// TIA Portal project "Organizador de Cajas" (V18)

(* hardware
DEVICE "S7-1200 station_1"  S7-1200 Station
   slot 0: "Rack_0"  S7-1200 Rack  Rack  V1.0
   slot 1: "PLC_1"  CPU 1212C DC/DC/Rly  6ES7 212-1HE40-0XB0  V4.6
*)

// ===== PLC "PLC_1"  CPU 1212C DC/DC/Rly =====

VAR_GLOBAL   // PLC tag table "Default tag table"
   "pulsadorStart" AT %I0.0 : Bool;
   "pulsadorStop" AT %I0.1 : Bool;
   "setaEmergencia" AT %I0.2 : Bool;
   "infrarrojoEntradaCinta" AT %I0.3 : Bool;
   "infrarrojoPrimerDesviador" AT %I0.4 : Bool;
   "infrarrojoSegundoDesviador" AT %I0.5 : Bool;
   "infrarrojoTercerDesviador" AT %I0.6 : Bool;
   "marcaEnServicio" AT %M90.0 : Bool;
   "marcaPaqueteCinta" AT %M90.1 : Bool;
   "marcaTurnoDesviadorUno" AT %M90.2 : Bool;
   "marcaTurnoDesviadorDos" AT %M90.3 : Bool;
   "marcaTurnoDesviadorTres" AT %M90.4 : Bool;
   "ledStart" AT %Q0.0 : Bool;
   "ledStop" AT %Q0.1 : Bool;
   "motorCintaPrincipal" AT %Q0.2 : Bool;
   "desviadorUno" AT %Q0.3 : Bool;
   "cintaDesviadorUno" AT %Q0.4 : Bool;
   "desviadorDos" AT %Q0.5 : Bool;
   "cintaDesviadorDos" AT %Q0.6 : Bool;
   "desviadorTres" AT %Q0.7 : Bool;
   "cintaDesviadorTres" AT %Q1.0 : Bool;
END_VAR

// folder: System blocks/Program resources

DATA_BLOCK "retardoArranqueCinta"   // DB1
{ S7_Optimized_Access := 'TRUE' }
AUTHOR : Simatic
FAMILY : IEC
NAME : IEC_TMR
VERSION : 1.0
// stored: InstanceOfName IEC_TIMER
"IEC_TIMER"
BEGIN
END_DATA_BLOCK

DATA_BLOCK "cajaSeleccionada"   // DB2
{ S7_Optimized_Access := 'TRUE' }
AUTHOR : Simatic
FAMILY : IEC
NAME : IEC_TMR
VERSION : 1.0
// stored: InstanceOfName IEC_TIMER
"IEC_TIMER"
BEGIN
END_DATA_BLOCK

DATA_BLOCK "CTUDesviadorUno"   // DB3
{ S7_Optimized_Access := 'TRUE' }
AUTHOR : Simatic
FAMILY : IEC
NAME : CNTR
VERSION : 1.0
// stored: InstanceOfName IEC_COUNTER
"IEC_COUNTER"
BEGIN
END_DATA_BLOCK

DATA_BLOCK "CTUDesviadorDos"   // DB4
{ S7_Optimized_Access := 'TRUE' }
AUTHOR : Simatic
FAMILY : IEC
NAME : CNTR
VERSION : 1.0
// stored: InstanceOfName IEC_COUNTER
"IEC_COUNTER"
BEGIN
END_DATA_BLOCK

DATA_BLOCK "CTUDesviadorTres"   // DB5
{ S7_Optimized_Access := 'TRUE' }
AUTHOR : Simatic
FAMILY : IEC
NAME : CNTR
VERSION : 1.0
// stored: InstanceOfName IEC_COUNTER
"IEC_COUNTER"
BEGIN
END_DATA_BLOCK

// folder: (top level)

ORGANIZATION_BLOCK "Main"   // OB1, LAD, ProgramCycle
TITLE = "Main Program Sweep (Cycle)"
{ S7_Optimized_Access := 'TRUE' }
VERSION : 0.1
   VAR_INPUT
      Initial_Call : Bool;   // Initial call of this OB
      Remanence : Bool;   // =True, if remanent data are available
   END_VAR
BEGIN

REGION Network 1: Instalación activa
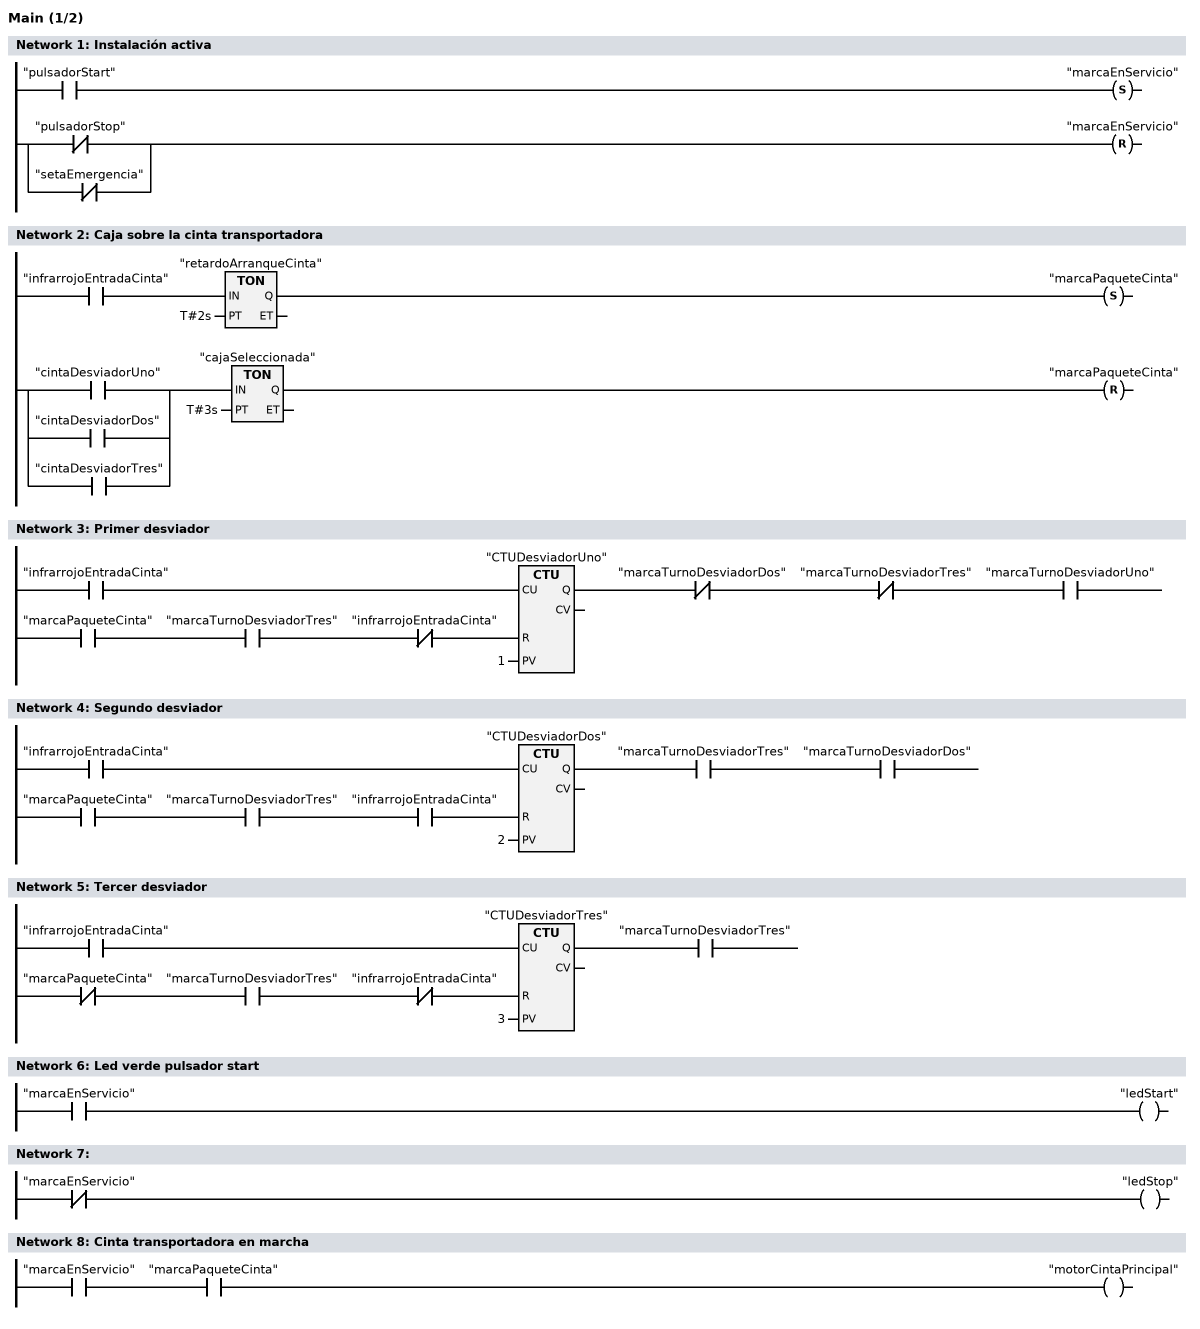
   RUNG wire#powerrail
      Contact( "pulsadorStart" )
      S_Coil( "marcaEnServicio" )
   END_RUNG
   RUNG wire#powerrail
      I_Contact( "pulsadorStop" )
      wire#w1
      R_Coil( "marcaEnServicio" )
   END_RUNG
   RUNG wire#powerrail
      I_Contact( "setaEmergencia" )
   END_RUNG wire#w1
   // the same network as SCL:
   IF "pulsadorStart" THEN "marcaEnServicio" := TRUE; END_IF;
   IF NOT "pulsadorStop" OR NOT "setaEmergencia" THEN "marcaEnServicio" := FALSE; END_IF;
END_REGION

REGION Network 2: Caja sobre la cinta transportadora
   "retardoArranqueCinta".TON(IN := "infrarrojoEntradaCinta", PT := T#2s);
   IF "retardoArranqueCinta".Q THEN "marcaPaqueteCinta" := TRUE; END_IF;
   "cajaSeleccionada".TON(IN := "cintaDesviadorUno" OR "cintaDesviadorDos" OR "cintaDesviadorTres", PT := T#3s);
   IF "cajaSeleccionada".Q THEN "marcaPaqueteCinta" := FALSE; END_IF;
END_REGION

REGION Network 3: Primer desviador
   "CTUDesviadorUno".CTU(CU := "infrarrojoEntradaCinta",
                         R := "marcaPaqueteCinta" AND "marcaTurnoDesviadorTres" AND NOT "infrarrojoEntradaCinta",
                         PV := 1);
END_REGION

REGION Network 4: Segundo desviador
   "CTUDesviadorDos".CTU(CU := "infrarrojoEntradaCinta",
                         R := "marcaPaqueteCinta" AND "marcaTurnoDesviadorTres" AND "infrarrojoEntradaCinta",
                         PV := 2);
END_REGION

REGION Network 5: Tercer desviador
   "CTUDesviadorTres".CTU(CU := "infrarrojoEntradaCinta",
                          R := NOT "marcaPaqueteCinta" AND "marcaTurnoDesviadorTres" AND NOT "infrarrojoEntradaCinta",
                          PV := 3);
END_REGION

REGION Network 6: Led verde pulsador start
   RUNG wire#powerrail
      Contact( "marcaEnServicio" )
      Coil( "ledStart" )
   END_RUNG
   // the same network as SCL:
   "ledStart" := "marcaEnServicio";
END_REGION

REGION Network 7
   RUNG wire#powerrail
      I_Contact( "marcaEnServicio" )
      Coil( "ledStop" )
   END_RUNG
   // the same network as SCL:
   "ledStop" := NOT "marcaEnServicio";
END_REGION

REGION Network 8: Cinta transportadora en marcha
   RUNG wire#powerrail
      Contact( "marcaEnServicio" )
      Contact( "marcaPaqueteCinta" )
      Coil( "motorCintaPrincipal" )
   END_RUNG
   // the same network as SCL:
   "motorCintaPrincipal" := "marcaEnServicio" AND "marcaPaqueteCinta";
END_REGION

REGION Network 9: Desviador uno abierto (accionado) + cinta en marcha
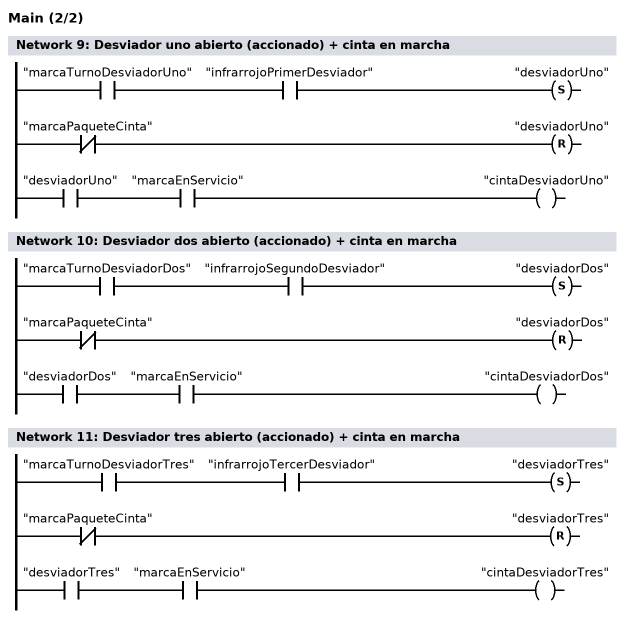
   RUNG wire#powerrail
      Contact( "marcaTurnoDesviadorUno" )
      Contact( "infrarrojoPrimerDesviador" )
      S_Coil( "desviadorUno" )
   END_RUNG
   RUNG wire#powerrail
      I_Contact( "marcaPaqueteCinta" )
      R_Coil( "desviadorUno" )
   END_RUNG
   RUNG wire#powerrail
      Contact( "desviadorUno" )
      Contact( "marcaEnServicio" )
      Coil( "cintaDesviadorUno" )
   END_RUNG
   // the same network as SCL:
   IF "marcaTurnoDesviadorUno" AND "infrarrojoPrimerDesviador" THEN "desviadorUno" := TRUE; END_IF;
   IF NOT "marcaPaqueteCinta" THEN "desviadorUno" := FALSE; END_IF;
   "cintaDesviadorUno" := "desviadorUno" AND "marcaEnServicio";
END_REGION

REGION Network 10: Desviador dos abierto (accionado) + cinta en marcha
   RUNG wire#powerrail
      Contact( "marcaTurnoDesviadorDos" )
      Contact( "infrarrojoSegundoDesviador" )
      S_Coil( "desviadorDos" )
   END_RUNG
   RUNG wire#powerrail
      I_Contact( "marcaPaqueteCinta" )
      R_Coil( "desviadorDos" )
   END_RUNG
   RUNG wire#powerrail
      Contact( "desviadorDos" )
      Contact( "marcaEnServicio" )
      Coil( "cintaDesviadorDos" )
   END_RUNG
   // the same network as SCL:
   IF "marcaTurnoDesviadorDos" AND "infrarrojoSegundoDesviador" THEN "desviadorDos" := TRUE; END_IF;
   IF NOT "marcaPaqueteCinta" THEN "desviadorDos" := FALSE; END_IF;
   "cintaDesviadorDos" := "desviadorDos" AND "marcaEnServicio";
END_REGION

REGION Network 11: Desviador tres abierto (accionado) + cinta en marcha
   RUNG wire#powerrail
      Contact( "marcaTurnoDesviadorTres" )
      Contact( "infrarrojoTercerDesviador" )
      S_Coil( "desviadorTres" )
   END_RUNG
   RUNG wire#powerrail
      I_Contact( "marcaPaqueteCinta" )
      R_Coil( "desviadorTres" )
   END_RUNG
   RUNG wire#powerrail
      Contact( "desviadorTres" )
      Contact( "marcaEnServicio" )
      Coil( "cintaDesviadorTres" )
   END_RUNG
   // the same network as SCL:
   IF "marcaTurnoDesviadorTres" AND "infrarrojoTercerDesviador" THEN "desviadorTres" := TRUE; END_IF;
   IF NOT "marcaPaqueteCinta" THEN "desviadorTres" := FALSE; END_IF;
   "cintaDesviadorTres" := "desviadorTres" AND "marcaEnServicio";
END_REGION
END_ORGANIZATION_BLOCK